Staubli VAL3: template.pgx

program main()
begin
  close(tCurrentTool)
  pPointRx.config.shoulder = lefty
  pPointRx.config.elbow = epositive
  pPointRx.config.wrist = wpositive
  pPointRx2.config.shoulder = lefty
  pPointRx2.config.elbow = epositive
  pPointRx2.config.wrist = wpositive
  mCurrentSpeed.tvel = 100.00
  mCurrentSpeed.blend = joint
  mCurrentSpeed.reach = 0.010
  mCurrentSpeed.leave = 0.010
  // Program start
  mCurrentSpeed.tvel = 200.000
{}

  waitEndMove()
  // Program end

end
